FUNCTION SPLIT_LWORD_INTO_BYTES (* this Function extracts the 8 BYTES from a lword *)
  (* Standard: 61499-1; Description: Copyright (c) 2026 HR Agrartechnik GmbH This program and the accompanying materials are made available under the terms of the Eclipse Public License 2.0 which is available at https://www.eclipse.org/legal/epl-2.0/ SPDX-License-Identifier: EPL-2.0 *)
  (* Version 1.0, 2026-05-16, Franz Höpfinger, HR Agrartechnik, initial Implementation *)
  PACKAGE eclipse4diac::utils::splitting;
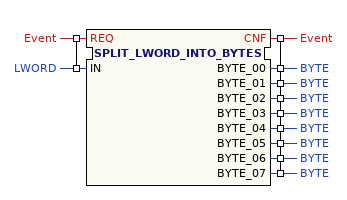
  EVENT_INPUT
    REQ WITH IN; (* Normal Execution Request *)
  END_EVENT
  EVENT_OUTPUT
    CNF WITH BYTE_00, BYTE_01, BYTE_02, BYTE_03, BYTE_04, BYTE_05, BYTE_06, BYTE_07; (* Execution Confirmation *)
  END_EVENT
  VAR_INPUT
    IN : LWORD;
  END_VAR
  VAR_OUTPUT
    BYTE_00 : BYTE;
    BYTE_01 : BYTE;
    BYTE_02 : BYTE;
    BYTE_03 : BYTE;
    BYTE_04 : BYTE;
    BYTE_05 : BYTE;
    BYTE_06 : BYTE;
    BYTE_07 : BYTE;
  END_VAR
  BODY IN ST:
(* this Function extracts the 8 BYTES from a lword *)
FUNCTION SPLIT_LWORD_INTO_BYTES

VAR_INPUT
	IN : LWORD;
END_VAR

VAR_OUTPUT
	BYTE_00 : BYTE;
	BYTE_01 : BYTE;
	BYTE_02 : BYTE;
	BYTE_03 : BYTE;
	BYTE_04 : BYTE;
	BYTE_05 : BYTE;
	BYTE_06 : BYTE;
	BYTE_07 : BYTE;
END_VAR

BYTE_00 := IN.%B0;
BYTE_01 := IN.%B1;
BYTE_02 := IN.%B2;
BYTE_03 := IN.%B3;
BYTE_04 := IN.%B4;
BYTE_05 := IN.%B5;
BYTE_06 := IN.%B6;
BYTE_07 := IN.%B7;

END_FUNCTION
  END_BODY
END_FUNCTION
